// TwinCAT 3 PLC project HelloWorld
// ProgramVersion: 3.1.4024.0
// libraries:
//   Tc2_Standard, * (Beckhoff Automation GmbH)
//   Tc2_System, * (Beckhoff Automation GmbH)
//   Tc2_Utilities, * (Beckhoff Automation GmbH)
//   Tc3_Module, * (Beckhoff Automation GmbH)
// project tree:
//   DUTs/ E_Color.TcDUT (not stored), E_Event.TcDUT (not stored), ST_Event.TcDUT (not stored), ST_Student.TcDUT (not stored)
//   GVLs/ Nums.TcGVL (not stored)
//   / PlcTask.TcTTO, PlcTask_1.TcTTO (not stored)
//   POUs/ Celcius_Fahrenheit.TcPOU (not stored), F_Add.TcPOU (not stored), F_InitializeStudentDetails.TcPOU, F_Loops.TcPOU (not stored), F_Multiply.TcPOU (not stored), F_PrimeCheck.TcPOU (not stored), F_UpdateTimeWithSystemTime.TcPOU (not stored), F_HelloWorld.TcPOU (not stored), MAIN.TcPOU, My_Program.TcPOU (not stored)
// real-time tasks:
//   TASK PlcTask: cycle T#10ms, priority 1, ADS port 350
//   TASK PlcTask_1: cycle T#10ms, priority 20, ADS port 351

CONFIGURATION HelloWorld
    RESOURCE PLC ON TwinCAT3
        TASK PlcTask(INTERVAL := T#10ms, PRIORITY := 20);
        PROGRAM MAIN WITH PlcTask : MAIN;
    END_RESOURCE
END_CONFIGURATION

// ---- POUs/MAIN.TcPOU
PROGRAM MAIN
VAR
	fFahrenheit : REAL;
	stEventOne : ST_Event;
	bFlag : BOOL := FALSE;
	nSum : INT;
	nProd : DINT;
	bIsPrime : BOOL;
	nResultFromLoop1 : INT;
	nResultFromLoop2 : INT;
	nResultFromLoop3 : INT;
	nNum1 :INT := 22;
	
	stStudentReference1 : ST_Student;
END_VAR


//IF NOT bFlag THEN 
fFahrenheit := Celcius_Fahrenheit(fCelcius := 5.0);
F_UpdateTimeWithSystemTime(stEventOne);
F_Add(nFirstNum:= nNum1, nSecondNum:= 32,nResult => nSum );
bFlag := TRUE;
nProd := F_Multiply(123,432);
bIsPrime := F_PrimeCheck(nInputNum := 17 );

F_InitializeStudentDetails(stStudentReference1, 'Kamesh', 101 , 21);

F_Loops(10,nResult1 => nResultFromLoop1, nResult2 => nResultFromLoop2, nResult3 => nResultFromLoop3);

//END_IF

END_PROGRAM

// ---- POUs/F_InitializeStudentDetails.TcPOU
FUNCTION F_InitializeStudentDetails
VAR_INPUT
	stStudent1 : REFERENCE TO ST_Student;
	stName : STRING(255);
	stId : INT;
	stAge :INT;
END_VAR
VAR
END_VAR

stStudent1.sStudentName := stName;
stStudent1.nStudentAge := stAge;
stStudent1.nStudentId := stStudent1.nStudentId + stId;

END_FUNCTION
